// TIA Portal V20 export
TYPE "typeSequenceControlNodeJobInterfaceMonitoring"
// stored: Namespace Unit1.Em6
   STRUCT
      busyVisionInspection { ExternalWritable := 'False'} : Bool;
      doneVisionInspection { ExternalWritable := 'False'} : Bool;
   END_STRUCT;
END_TYPE
